(* IEC 61131-3 sources: plc-projects/02-latch-circuit/build, 2 files *)

(* ---- plc.st ---- *)
TYPE
  LOGLEVEL : (CRITICAL, WARNING, INFO, DEBUG) := INFO;
END_TYPE

FUNCTION_BLOCK LOGGER
  VAR_INPUT
    TRIG : BOOL;
    MSG : STRING;
    LEVEL : LOGLEVEL := INFO;
  END_VAR
  VAR
    TRIG0 : BOOL;
  END_VAR

  IF TRIG AND NOT TRIG0 THEN
  {{
   LogMessage(GetFbVar(LEVEL),(char*)GetFbVar(MSG, .body),GetFbVar(MSG, .len));
  }}
  END_IF;
  TRIG0:=TRIG;
END_FUNCTION_BLOCK

PROGRAM program2
  VAR
    Start AT %IX0.1 : BOOL;
    Stop AT %IX0.2 : BOOL;
    LED AT %QX0.1 : BOOL;
  END_VAR

  LED := NOT(Stop) AND (LED OR Start);
END_PROGRAM

CONFIGURATION Config0

  RESOURCE Res0 ON PLC
    TASK task0(INTERVAL := T#20ms,PRIORITY := 0);
    PROGRAM instance0 WITH task0 : program2;
  END_RESOURCE
END_CONFIGURATION

(* ---- generated_plc.st ---- *)
PROGRAM program2
  VAR
    Start AT %IX0.1 : BOOL;
    Stop AT %IX0.2 : BOOL;
    LED AT %QX0.1 : BOOL;
  END_VAR

  LED := NOT(Stop) AND (LED OR Start);
END_PROGRAM

CONFIGURATION Config0

  RESOURCE Res0 ON PLC
    TASK task0(INTERVAL := T#20ms,PRIORITY := 0);
    PROGRAM instance0 WITH task0 : program2;
  END_RESOURCE
END_CONFIGURATION
